# EPICS substitutions: iocBoot/iocbcur/pydevice_scripts.substitutions
file "user_python_script.db"
{
pattern
{N}
{1}
{2}
{3}
{4}
{5}
}
